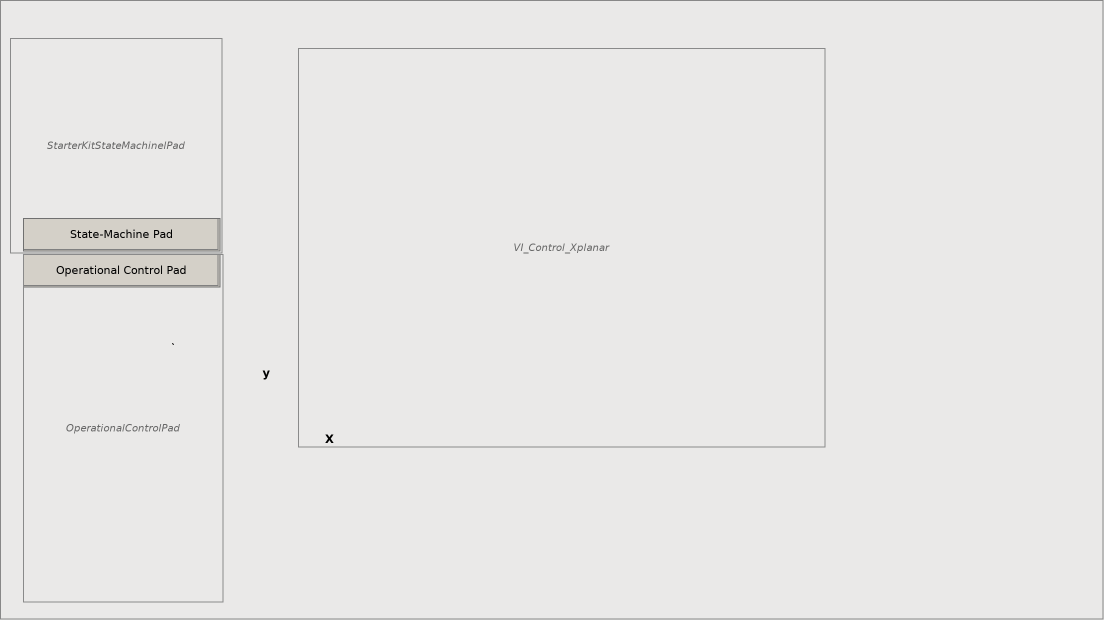
VISUALIZATION VI_MainSide  // 1104x620
    Polygon (172,343) (173,344)
    Frame (298,48 527x399)
        shows VI_Control_Xplanar()
    Label (316,424 27x30), "X"
    Label (253,358 27x30), "y"
    Button (23,254 197x33), "Operational Control Pad", invisible if: NOT stVisControl.stOperatorPad.bVisInvisible
        p3560616238: stVisControl.stOperatorPad.nButtonPositionX
        p2738717112: stVisControl.stOperatorPad.nButtonPositionY
        OnMouseClick: execute { stVisControl.stOperatorPad.bVisInvisibleButton := FALSE; }
    Button (23,218 197x33), "State-Machine Pad", invisible if: NOT stVisControl.stControlPad.bVisInvisible
        p3560616238: stVisControl.stControlPad.nButtonPositionX
        p2738717112: stVisControl.stControlPad.nButtonPositionY
        OnMouseClick: execute { stVisControl.stControlPad.bVisInvisibleButton := FALSE; }
    Frame (10,38 212x215), invisible if: stVisControl.stControlPad.bVisInvisible
        shows StarterKitStateMachinelPad(stControlPadControl := stVisControl.stControlPad)
        p3560616238: stVisControl.stControlPad.nFramePositionX
        p2738717112: stVisControl.stControlPad.nFramePositionY
    Frame (23,254 200x348), invisible if: stVisControl.stOperatorPad.bVisInvisible
        shows OperationalControlPad(stVisOperationalControl := stVisControl.stOperatorPad)
        p3560616238: stVisControl.stOperatorPad.nFramePositionX
        p2738717112: stVisControl.stOperatorPad.nFramePositionY
END_VISUALIZATION

(* stored: Version 1.1.0.1, ProductVersion 3.1.4024.9
   Visu VI_MainSide: Id {c9ec1629-9532-44ea-8cb4-f2ecd996ba5c} *)
